FUNCTION_BLOCK FB_ReadTc3Events2 EXTENDS FB_ReadTc3Events
VAR_INPUT
	bClearLoggedTable	:BOOL;
END_VAR
VAR_OUTPUT
	LoggedEvents: ARRAY [1..200] OF ST_ReadEventW;
END_VAR

SUPER^();

IF bClearLoggedTable THEN
	MEMSET(ADR(LoggedEvents),0,SIZEOF(LoggedEvents));
END_IF

METHOD ReadLoggedEvents : HRESULT
VAR_INPUT
END_VAR
END_METHOD

END_FUNCTION_BLOCK

(* stored: Version 1.1.0.1
   POU FB_ReadTc3Events2: Id {5a6edfd8-5abe-4422-80aa-514948601d1b}, SpecialFunc None
   Method ReadLoggedEvents: Id {936688d8-92ba-4ae8-8c66-ec3f8ec0b489} *)
